// TwinCAT 3 PLC project LogHandler
// Title: Log Handler
// Company: Marden Edwards
// Author: Piotr Pawlowski
// ProjectVersion: 1.0.0.0
// ProgramVersion: 3.1.4026.19
// libraries:
//   Tc2_Standard, * (Beckhoff Automation GmbH)
//   Tc2_System, * (Beckhoff Automation GmbH)
//   Tc2_Utilities, * (Beckhoff Automation GmbH)
// project tree:
//   DUTs/LogData/ ST_EventData.TcDUT
//   DUTs/String/ libT_LongSTRING.TcDUT
//   POUs/Logger FBs/ FB_EventHandler.TcPOU
//   Version/ Global_Version.TcGVL
// real-time tasks:
//   TASK TcUnit_Task: cycle T#10ms, priority 10, ADS port 350

// ---- DUTs/LogData/ST_EventData.TcDUT
TYPE ST_EventData :
STRUCT
	bEnable					: BOOL;
	nCounter				: UDINT;
	sTimeStamp				: STRING;
	nImageByte				: UINT;
	aDataLogImage			: ARRAY[0..65000] OF BYTE;
	nMaxImageArraySize		: UINT := 65000 ;
	nControlSize			: UINT;
	bBufferOverflow			: BOOL;
END_STRUCT
END_TYPE

// ---- DUTs/String/libT_LongSTRING.TcDUT
TYPE libT_LongSTRING : STRING(1023);
END_TYPE

// ---- Version/Global_Version.TcGVL
{attribute 'TcGenerated'}
{attribute 'no-analysis'}
{attribute 'linkalways'}
// This function has been automatically generated from the project information.
VAR_GLOBAL CONSTANT
	{attribute 'const_non_replaced'}
	stLibVersion_Log_Handler : ST_LibVersion := (iMajor := 1, iMinor := 0, iBuild := 0, iRevision := 0, nFlags := 0, sVersion := '1.0.0.0');
END_VAR

// ---- POUs/Logger FBs/FB_EventHandler.TcPOU
FUNCTION_BLOCK FB_EventHandler
VAR_INPUT
	_IsUsed					: BOOL;
	bLogData					: BOOL;
	sLogMessage				: libT_LongSTRING;
END_VAR
VAR_IN_OUT
	stEventData				: ST_EventData;
END_VAR
VAR_OUTPUT
	bDone						: BOOL;
	bBufferOverflow			: BOOL;
END_VAR
VAR
	rtExecute					: R_TRIG;
	sString 					: libT_LongSTRING;
	nStringLen					: UINT;

END_VAR

_IsUsed := TRUE;

rtExecute(CLK:=bLogData);

IF NOT stEventData.bBufferOverflow AND stEventData.bEnable AND sLogMessage <> '' AND rtExecute.Q THEN

	sString := '';
	(*stEventData.nCounter := stEventData.nCounter + 1;
	sString := F_CONCAT4(F_AddPaddingUDINT(stEventData.nCounter, 7), ' : ', stEventData.sTimeStamp, ' : ');*)
	//sString := CONCAT(stEventData.sTimeStamp, ' : ');
	//sString := F_LongCONCAT(sString,sLogMessage);
	//sString := F_LongCONCAT(sString,'.$R$N');
	CONCAT2(ADR(stEventData.sTimeStamp), ADR(' : '), ADR(sString), SIZEOF(sString));
	CONCAT2(ADR(sString), ADR(sLogMessage), ADR(sString), SIZEOF(sString));
	CONCAT2(ADR(sString), ADR('.$R$N'), ADR(sString), SIZEOF(sString));
	nStringLen := TO_UINT(LEN2(ADR(sString)));  //Max size 1024 byte -> LongString

	stEventData.nControlSize := stEventData.nControlSize + nStringLen;

	IF stEventData.nControlSize <  stEventData.nMaxImageArraySize THEN
		MEMMOVE(ADR(stEventData.aDataLogImage[stEventData.nImageByte]), ADR(sString), nStringLen);
		stEventData.nImageByte := stEventData.nImageByte + nStringLen;
	ELSE
		stEventData.bBufferOverflow	:=TRUE;
		bBufferOverflow	:= TRUE;
	END_IF

	bDone	:= TRUE;
	(*F_LOG_Handler := TRUE;*)
ELSE
	bDone	:= FALSE;
END_IF

END_FUNCTION_BLOCK
